TYPE hw_button_location:
    (Released_hw_button_location, Pushed_hw_button_location);
END_TYPE

(* stored: ProductVersion 3.1.0.18, Version 1.1.0.1 *)
